TYPE E_StepEndCause : (
    STEP_END_NONE := 0,
    STEP_END_PRIMARY_RELATIVE_DISTANCE := 10,
    STEP_END_PRIMARY_STEP_TIME := 20,
    STEP_END_PRIMARY_FORCE_DECLINE := 30,
    STEP_END_SECONDARY_RELATIVE_DISTANCE := 40,
    STEP_END_MAX_TIME := 50,
    STEP_END_HARD_FORCE := 60,
    STEP_END_HARD_STROKE := 70,
    STEP_END_COLLISION := 110,
    STEP_END_SENSOR_INVALID := 80,
    STEP_END_AXIS_FAULT := 90,
    STEP_END_STOP_REQUEST := 100
); END_TYPE

(* stored: Version 1.1.0.1
   DUT E_StepEndCause: Id {E3000000-0000-4000-8000-000000000012} *)
